// TIA Portal V17 export
// export: Created 2024-08-07T21:44:00.5183403Z, ExportSetting WithDefaults, DisplayName Totally Integrated Automation Portal, DisplayVersion V17 Update 7, DisplayName TIA Portal Openness, DisplayVersion V17 Update 7, DisplayName TIA Portal Version Control Interface, DisplayVersion V17, DisplayName SINAMICS Startdrive Advanced, DisplayVersion V17 SP2, DisplayName SINAMICS Startdrive G110M, G120, G120C, G120D, G120P, G115D, DisplayVersion V17 SP2, DisplayName SINAMICS Startdrive G130, G150, S120, S150, SINAMICS MV, S210, DisplayVersion V17 SP2, DisplayName STEP 7 Professional, DisplayVersion V17 Update 7, DisplayName STEP 7 Safety, DisplayVersion V17 Update 6, DisplayName WinCC Advanced / Unified PC, DisplayVersion V17 Update 7
FUNCTION_BLOCK "FB_DateTimeAndShifts"   // FB5010, LAD
{ S7_Optimized_Access := 'TRUE' }
VERSION : 0.1
// stored: AutoNumber false, IsIECCheckEnabled false, IsRetainMemResEnabled false, MemoryReserve 100, SetENOAutomatically false, UDAEnableTagReadback false
   VAR_INPUT
      iSettingsSecurity : Bool;
   END_VAR
   VAR
      Edges : Struct
         Shift1Started : Bool;
         Shift2Started : Bool;
         Shift3Started : Bool;
      END_STRUCT;
   END_VAR
   VAR RETAIN
      Settings : Struct
         Actual { S7_SetPoint := 'True'} : "UDT_DateTimeAndShiftsSettings";
         Last { S7_SetPoint := 'True'} : "UDT_DateTimeAndShiftsSettings";
         Status : Struct
            SettingsCanBeChanged : Bool;   // 0= No
         END_STRUCT;
         Commands : Struct
            DateAndTimeUse : Bool;
            DateAndTimeSet : Bool;
         END_STRUCT;
      END_STRUCT;
   END_VAR
   VAR
      ActualValues : Struct
         DateAndTime : DTL;
         DayOfYear : UInt;
      END_STRUCT;
      ShiftStatus { S7_SetPoint := 'True'} : "UDT_ShiftStatus";
      TimeTransformationRule { S7_SetPoint := 'True'} : TimeTransformationRule;
      Set_timezone_results { ExternalAccessible := 'False'; ExternalVisible := 'False'; ExternalWritable := 'False'} : Struct
         done { ExternalAccessible := 'False'; ExternalVisible := 'False'; ExternalWritable := 'False'} : Bool;
         busy { ExternalAccessible := 'False'; ExternalVisible := 'False'; ExternalWritable := 'False'} : Bool;
         error { ExternalAccessible := 'False'; ExternalVisible := 'False'; ExternalWritable := 'False'} : Bool;
         status { ExternalAccessible := 'False'; ExternalVisible := 'False'; ExternalWritable := 'False'} : Word;
      END_STRUCT;
   END_VAR
   VAR_TEMP
      i : Int;
      ui : UInt;
      actual_time : Time_Of_Day;
      dst : Bool;
   END_VAR
   VAR_TEMP   // added for the SCL form of the ladder/FBD networks
      _w1 : Bool;
      _w2 : Bool;
      _w3 : Bool;
      _w4 : Bool;
      _w5 : Bool;
      _w6 : Bool;
      _w7 : Bool;
      _w8 : Bool;
   END_VAR
BEGIN

REGION Network 1 (SCL)
   #TimeTransformationRule.Bias := -360;
   #TimeTransformationRule.DaylightBias := 0;
   #TimeTransformationRule.DaylightStartMonth := 3;
   #TimeTransformationRule.DaylightStartWeek := 5;
   #TimeTransformationRule.DaylightStartWeekday := 1;
   #TimeTransformationRule.DaylightStartHour := 2;
   #TimeTransformationRule.DaylightStartMinute := 0;
   #TimeTransformationRule.StandardStartMonth := 10;
   #TimeTransformationRule.StandardStartWeek := 5;
   #TimeTransformationRule.StandardStartWeekday := 1;
   #TimeTransformationRule.StandardStartHour := 3;
   #TimeTransformationRule.StandardStartMinute := 0;
END_REGION

REGION Network 2: Settings control
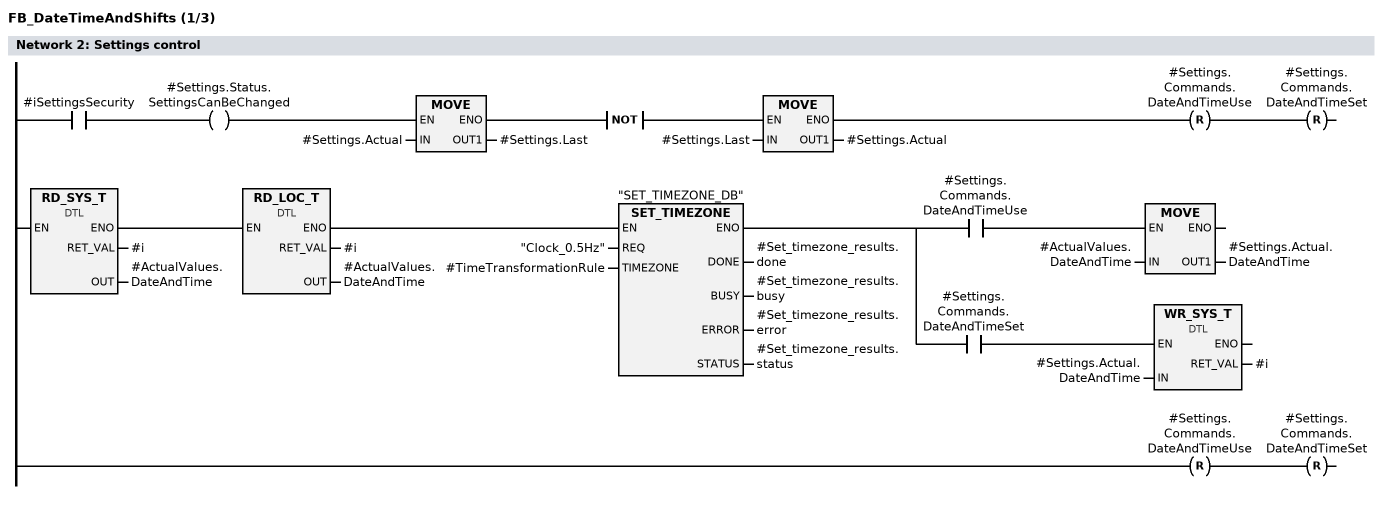
   RUNG wire#powerrail
      Contact( #iSettingsSecurity )
      Coil( #Settings.Status.SettingsCanBeChanged )
      Move(in := #Settings.Actual, out1 => #Settings.Last)
      Not()
      Move(in := #Settings.Last, out1 => #Settings.Actual)
      R_Coil( #Settings.Commands.DateAndTimeUse )
      R_Coil( #Settings.Commands.DateAndTimeSet )
   END_RUNG
   RUNG wire#powerrail
      { S7_Templates := "date_type := DTL" } RD_SYS_T(RET_VAL => #i, OUT => #ActualValues.DateAndTime)
      { S7_Templates := "date_type := DTL" } RD_LOC_T(RET_VAL => #i, OUT => #ActualValues.DateAndTime)
      "SET_TIMEZONE_DB".SET_TIMEZONE(REQ := "Clock_0.5Hz", TimeZone := #TimeTransformationRule, DONE => #Set_timezone_results.done, BUSY => #Set_timezone_results.busy, ERROR => #Set_timezone_results.error, STATUS => #Set_timezone_results.status)
      wire#w1
      Contact( #Settings.Commands.DateAndTimeUse )
      Move(in := #ActualValues.DateAndTime, out1 => #Settings.Actual.DateAndTime)
   END_RUNG
   RUNG wire#w1
      Contact( #Settings.Commands.DateAndTimeSet )
      { S7_Templates := "date_type := DTL" } WR_SYS_T(IN := #Settings.Actual.DateAndTime, RET_VAL => #i)
   END_RUNG
   RUNG wire#powerrail
      R_Coil( #Settings.Commands.DateAndTimeUse )
      R_Coil( #Settings.Commands.DateAndTimeSet )
   END_RUNG
   // the same network as SCL:
   #Settings.Status.SettingsCanBeChanged := #iSettingsSecurity;
   IF #iSettingsSecurity THEN #Settings.Last := #Settings.Actual; END_IF;
   IF NOT #iSettingsSecurity THEN
       #Settings.Actual := #Settings.Last;
       #Settings.Commands.DateAndTimeUse := FALSE;
       #Settings.Commands.DateAndTimeSet := FALSE;
   END_IF;
   #i := RD_SYS_T(OUT => #ActualValues.DateAndTime, ENO => #_w1);
   #i := RD_LOC_T(EN := #_w1, OUT => #ActualValues.DateAndTime, ENO => #_w2);
   "SET_TIMEZONE_DB"(EN := #_w2,   // SET_TIMEZONE
                     REQ := "Clock_0.5Hz",
                     TimeZone := #TimeTransformationRule,
                     DONE => #Set_timezone_results.done,
                     BUSY => #Set_timezone_results.busy,
                     ERROR => #Set_timezone_results.error,
                     STATUS => #Set_timezone_results.status,
                     ENO => #_w3);
   IF #_w3 AND #Settings.Commands.DateAndTimeUse THEN
       #Settings.Actual.DateAndTime := #ActualValues.DateAndTime;
   END_IF;
   IF #_w3 AND #Settings.Commands.DateAndTimeSet THEN
       #i := WR_SYS_T(IN := #Settings.Actual.DateAndTime);
   END_IF;
   #Settings.Commands.DateAndTimeUse := FALSE;
   #Settings.Commands.DateAndTimeSet := FALSE;
END_REGION

REGION Network 3: Day of year
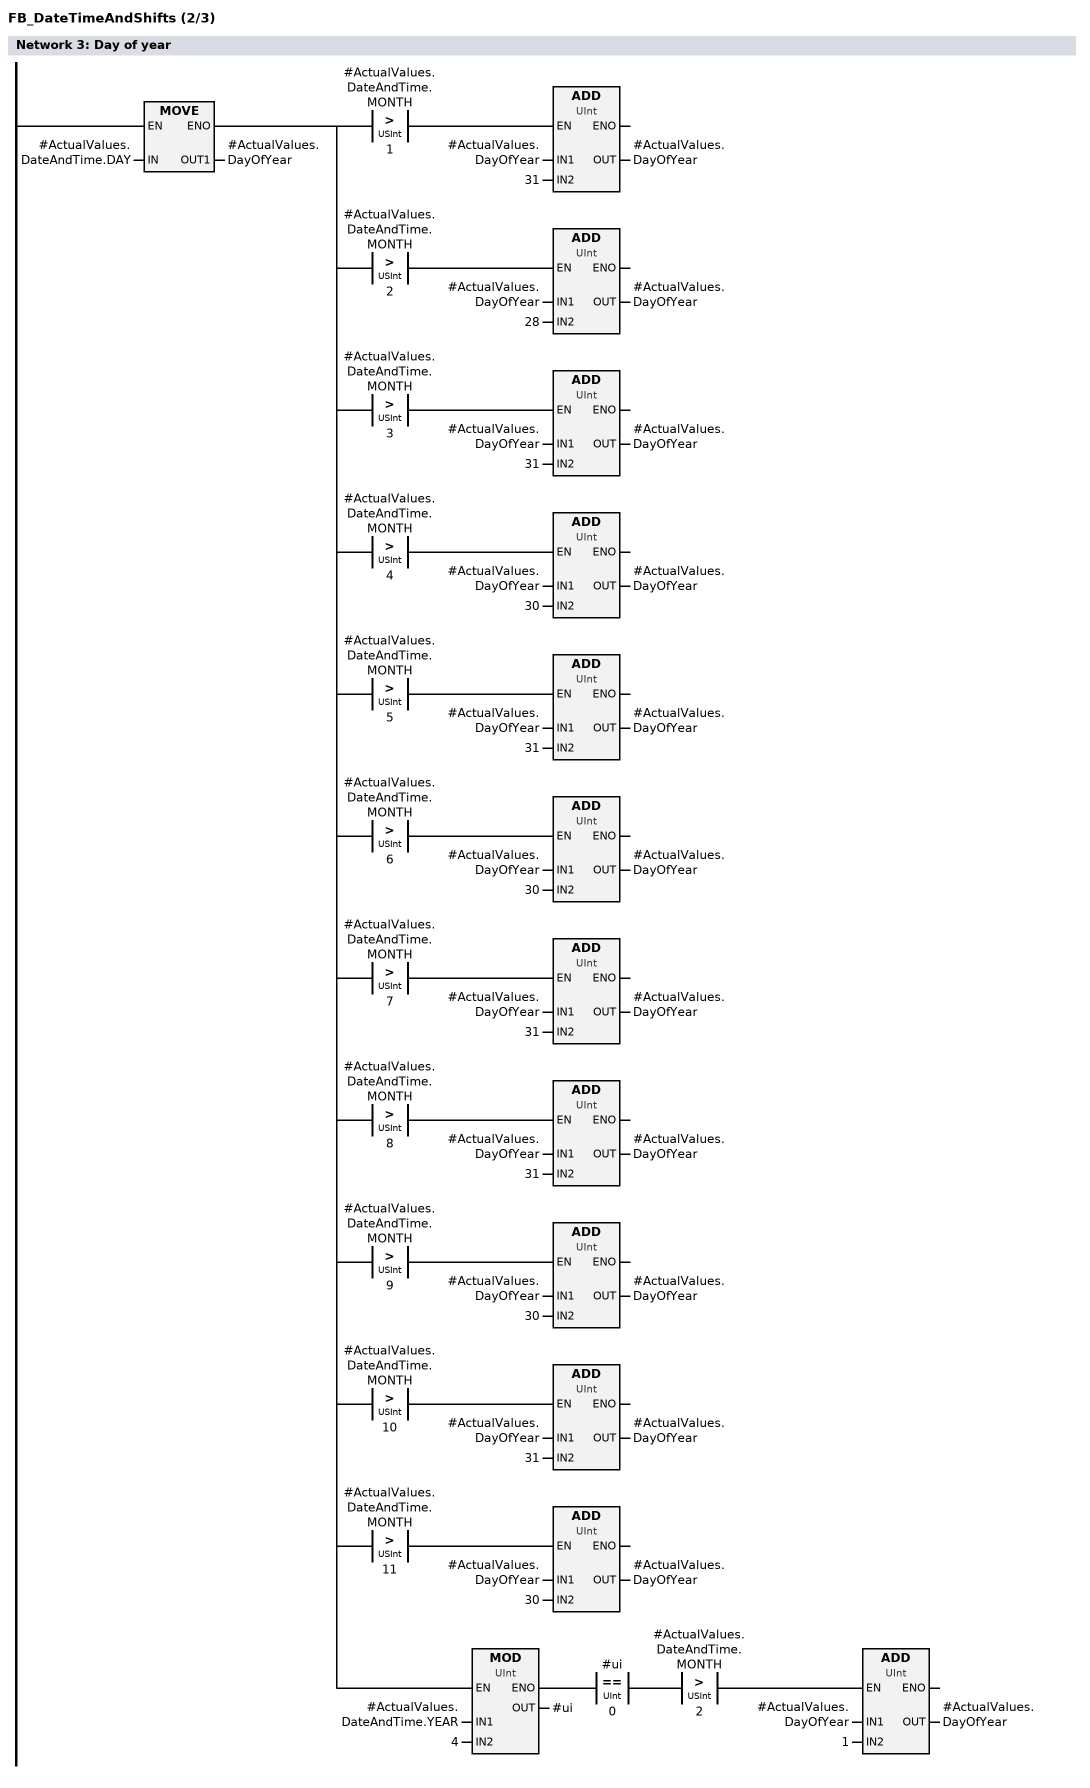
   RUNG wire#powerrail
      Move(in := #ActualValues.DateAndTime.DAY, out1 => #ActualValues.DayOfYear)
      wire#w1
      { S7_Templates := "SrcType := USInt" } GT_Contact(in1 := #ActualValues.DateAndTime.MONTH, in2 := 1)
      { S7_Templates := "SrcType := UInt" } Add(in1 := #ActualValues.DayOfYear, in2 := 31, out => #ActualValues.DayOfYear)
   END_RUNG
   RUNG wire#w1
      { S7_Templates := "SrcType := USInt" } GT_Contact(in1 := #ActualValues.DateAndTime.MONTH, in2 := 2)
      { S7_Templates := "SrcType := UInt" } Add(in1 := #ActualValues.DayOfYear, in2 := 28, out => #ActualValues.DayOfYear)
   END_RUNG
   RUNG wire#w1
      { S7_Templates := "SrcType := USInt" } GT_Contact(in1 := #ActualValues.DateAndTime.MONTH, in2 := 3)
      { S7_Templates := "SrcType := UInt" } Add(in1 := #ActualValues.DayOfYear, in2 := 31, out => #ActualValues.DayOfYear)
   END_RUNG
   RUNG wire#w1
      { S7_Templates := "SrcType := USInt" } GT_Contact(in1 := #ActualValues.DateAndTime.MONTH, in2 := 4)
      { S7_Templates := "SrcType := UInt" } Add(in1 := #ActualValues.DayOfYear, in2 := 30, out => #ActualValues.DayOfYear)
   END_RUNG
   RUNG wire#w1
      { S7_Templates := "SrcType := USInt" } GT_Contact(in1 := #ActualValues.DateAndTime.MONTH, in2 := 5)
      { S7_Templates := "SrcType := UInt" } Add(in1 := #ActualValues.DayOfYear, in2 := 31, out => #ActualValues.DayOfYear)
   END_RUNG
   RUNG wire#w1
      { S7_Templates := "SrcType := USInt" } GT_Contact(in1 := #ActualValues.DateAndTime.MONTH, in2 := 6)
      { S7_Templates := "SrcType := UInt" } Add(in1 := #ActualValues.DayOfYear, in2 := 30, out => #ActualValues.DayOfYear)
   END_RUNG
   RUNG wire#w1
      { S7_Templates := "SrcType := USInt" } GT_Contact(in1 := #ActualValues.DateAndTime.MONTH, in2 := 7)
      { S7_Templates := "SrcType := UInt" } Add(in1 := #ActualValues.DayOfYear, in2 := 31, out => #ActualValues.DayOfYear)
   END_RUNG
   RUNG wire#w1
      { S7_Templates := "SrcType := USInt" } GT_Contact(in1 := #ActualValues.DateAndTime.MONTH, in2 := 8)
      { S7_Templates := "SrcType := UInt" } Add(in1 := #ActualValues.DayOfYear, in2 := 31, out => #ActualValues.DayOfYear)
   END_RUNG
   RUNG wire#w1
      { S7_Templates := "SrcType := USInt" } GT_Contact(in1 := #ActualValues.DateAndTime.MONTH, in2 := 9)
      { S7_Templates := "SrcType := UInt" } Add(in1 := #ActualValues.DayOfYear, in2 := 30, out => #ActualValues.DayOfYear)
   END_RUNG
   RUNG wire#w1
      { S7_Templates := "SrcType := USInt" } GT_Contact(in1 := #ActualValues.DateAndTime.MONTH, in2 := 10)
      { S7_Templates := "SrcType := UInt" } Add(in1 := #ActualValues.DayOfYear, in2 := 31, out => #ActualValues.DayOfYear)
   END_RUNG
   RUNG wire#w1
      { S7_Templates := "SrcType := USInt" } GT_Contact(in1 := #ActualValues.DateAndTime.MONTH, in2 := 11)
      { S7_Templates := "SrcType := UInt" } Add(in1 := #ActualValues.DayOfYear, in2 := 30, out => #ActualValues.DayOfYear)
   END_RUNG
   RUNG wire#w1
      { S7_Templates := "SrcType := UInt" } Mod(in1 := #ActualValues.DateAndTime.YEAR, in2 := 4, out => #ui)
      { S7_Templates := "SrcType := UInt" } EQ_Contact(in1 := #ui, in2 := 0)
      { S7_Templates := "SrcType := USInt" } GT_Contact(in1 := #ActualValues.DateAndTime.MONTH, in2 := 2)
      { S7_Templates := "SrcType := UInt" } Add(in1 := #ActualValues.DayOfYear, in2 := 1, out => #ActualValues.DayOfYear)
   END_RUNG
   // the same network as SCL:
   #ActualValues.DayOfYear := #ActualValues.DateAndTime.DAY;
   IF #ActualValues.DateAndTime.MONTH > 1 THEN
       #ActualValues.DayOfYear := #ActualValues.DayOfYear + 31;
   END_IF;
   IF #ActualValues.DateAndTime.MONTH > 2 THEN
       #ActualValues.DayOfYear := #ActualValues.DayOfYear + 28;
   END_IF;
   IF #ActualValues.DateAndTime.MONTH > 3 THEN
       #ActualValues.DayOfYear := #ActualValues.DayOfYear + 31;
   END_IF;
   IF #ActualValues.DateAndTime.MONTH > 4 THEN
       #ActualValues.DayOfYear := #ActualValues.DayOfYear + 30;
   END_IF;
   IF #ActualValues.DateAndTime.MONTH > 5 THEN
       #ActualValues.DayOfYear := #ActualValues.DayOfYear + 31;
   END_IF;
   IF #ActualValues.DateAndTime.MONTH > 6 THEN
       #ActualValues.DayOfYear := #ActualValues.DayOfYear + 30;
   END_IF;
   IF #ActualValues.DateAndTime.MONTH > 7 THEN
       #ActualValues.DayOfYear := #ActualValues.DayOfYear + 31;
   END_IF;
   IF #ActualValues.DateAndTime.MONTH > 8 THEN
       #ActualValues.DayOfYear := #ActualValues.DayOfYear + 31;
   END_IF;
   IF #ActualValues.DateAndTime.MONTH > 9 THEN
       #ActualValues.DayOfYear := #ActualValues.DayOfYear + 30;
   END_IF;
   IF #ActualValues.DateAndTime.MONTH > 10 THEN
       #ActualValues.DayOfYear := #ActualValues.DayOfYear + 31;
   END_IF;
   IF #ActualValues.DateAndTime.MONTH > 11 THEN
       #ActualValues.DayOfYear := #ActualValues.DayOfYear + 30;
   END_IF;
   #ui := #ActualValues.DateAndTime.YEAR MOD 4;
   IF (#ui = 0) AND (#ActualValues.DateAndTime.MONTH > 2) THEN
       #ActualValues.DayOfYear := #ActualValues.DayOfYear + 1;
   END_IF;
END_REGION

REGION Network 4: Shifts
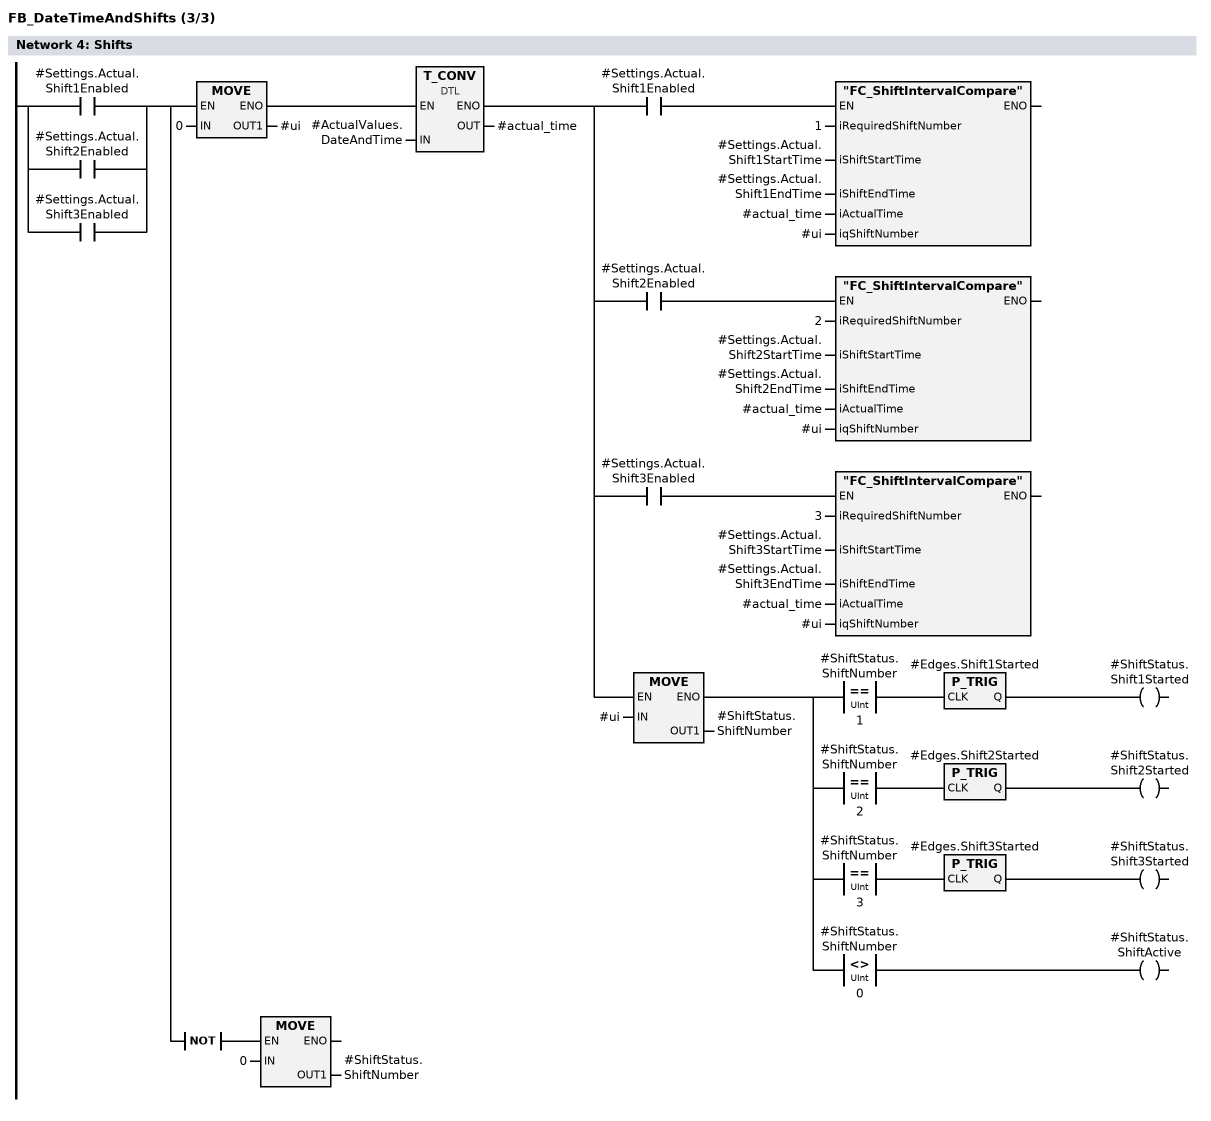
   RUNG wire#powerrail
      Contact( #Settings.Actual.Shift1Enabled )
      wire#w1
      Move(in := 0, out1 => #ui)
      { S7_Templates := "[src_type := DTL, dest_type := Time_Of_Day]" } T_CONV(IN := #ActualValues.DateAndTime, OUT => #actual_time)
      wire#w2
      Contact( #Settings.Actual.Shift1Enabled )
      "FC_ShiftIntervalCompare"(iRequiredShiftNumber := 1, iShiftStartTime := #Settings.Actual.Shift1StartTime, iShiftEndTime := #Settings.Actual.Shift1EndTime, iActualTime := #actual_time, iqShiftNumber := #ui)
   END_RUNG
   RUNG wire#powerrail
      Contact( #Settings.Actual.Shift2Enabled )
   END_RUNG wire#w1
   RUNG wire#powerrail
      Contact( #Settings.Actual.Shift3Enabled )
   END_RUNG wire#w1
   RUNG wire#w2
      Contact( #Settings.Actual.Shift2Enabled )
      "FC_ShiftIntervalCompare"(iRequiredShiftNumber := 2, iShiftStartTime := #Settings.Actual.Shift2StartTime, iShiftEndTime := #Settings.Actual.Shift2EndTime, iActualTime := #actual_time, iqShiftNumber := #ui)
   END_RUNG
   RUNG wire#w2
      Contact( #Settings.Actual.Shift3Enabled )
      "FC_ShiftIntervalCompare"(iRequiredShiftNumber := 3, iShiftStartTime := #Settings.Actual.Shift3StartTime, iShiftEndTime := #Settings.Actual.Shift3EndTime, iActualTime := #actual_time, iqShiftNumber := #ui)
   END_RUNG
   RUNG wire#w2
      Move(in := #ui, out1 => #ShiftStatus.ShiftNumber)
      wire#w3
      { S7_Templates := "SrcType := UInt" } EQ_Contact(in1 := #ShiftStatus.ShiftNumber, in2 := 1)
      P_Trig( #Edges.Shift1Started )
      Coil( #ShiftStatus.Shift1Started )
   END_RUNG
   RUNG wire#w3
      { S7_Templates := "SrcType := UInt" } EQ_Contact(in1 := #ShiftStatus.ShiftNumber, in2 := 2)
      P_Trig( #Edges.Shift2Started )
      Coil( #ShiftStatus.Shift2Started )
   END_RUNG
   RUNG wire#w3
      { S7_Templates := "SrcType := UInt" } EQ_Contact(in1 := #ShiftStatus.ShiftNumber, in2 := 3)
      P_Trig( #Edges.Shift3Started )
      Coil( #ShiftStatus.Shift3Started )
   END_RUNG
   RUNG wire#w3
      { S7_Templates := "SrcType := UInt" } NE_Contact(in1 := #ShiftStatus.ShiftNumber, in2 := 0)
      Coil( #ShiftStatus.ShiftActive )
   END_RUNG
   RUNG wire#w1
      Not()
      Move(in := 0, out1 => #ShiftStatus.ShiftNumber)
   END_RUNG
   // the same network as SCL:
   #_w1 := #Settings.Actual.Shift1Enabled OR #Settings.Actual.Shift2Enabled OR #Settings.Actual.Shift3Enabled;
   IF #_w1 THEN #ui := 0; END_IF;
   T_CONV(EN := #_w1, IN := #ActualValues.DateAndTime, OUT => #actual_time, ENO => #_w2);
   IF #_w2 AND #Settings.Actual.Shift1Enabled THEN
       "FC_ShiftIntervalCompare"(iRequiredShiftNumber := 1,
                               iShiftStartTime := #Settings.Actual.Shift1StartTime,
                               iShiftEndTime := #Settings.Actual.Shift1EndTime,
                               iActualTime := #actual_time,
                               iqShiftNumber := #ui);
   END_IF;
   IF #_w2 AND #Settings.Actual.Shift2Enabled THEN
       "FC_ShiftIntervalCompare"(iRequiredShiftNumber := 2,
                               iShiftStartTime := #Settings.Actual.Shift2StartTime,
                               iShiftEndTime := #Settings.Actual.Shift2EndTime,
                               iActualTime := #actual_time,
                               iqShiftNumber := #ui);
   END_IF;
   IF #_w2 AND #Settings.Actual.Shift3Enabled THEN
       "FC_ShiftIntervalCompare"(iRequiredShiftNumber := 3,
                               iShiftStartTime := #Settings.Actual.Shift3StartTime,
                               iShiftEndTime := #Settings.Actual.Shift3EndTime,
                               iActualTime := #actual_time,
                               iqShiftNumber := #ui);
   END_IF;
   IF #_w2 THEN #ShiftStatus.ShiftNumber := #ui; END_IF;
   #_w3 := #_w2 AND (#ShiftStatus.ShiftNumber = 1);
   #_w4 := #_w3 AND NOT #Edges.Shift1Started;   // rising edge
   #Edges.Shift1Started := #_w3;
   #ShiftStatus.Shift1Started := #_w4;
   #_w5 := #_w2 AND (#ShiftStatus.ShiftNumber = 2);
   #_w6 := #_w5 AND NOT #Edges.Shift2Started;   // rising edge
   #Edges.Shift2Started := #_w5;
   #ShiftStatus.Shift2Started := #_w6;
   #_w7 := #_w2 AND (#ShiftStatus.ShiftNumber = 3);
   #_w8 := #_w7 AND NOT #Edges.Shift3Started;   // rising edge
   #Edges.Shift3Started := #_w7;
   #ShiftStatus.Shift3Started := #_w8;
   #ShiftStatus.ShiftActive := #_w2 AND (#ShiftStatus.ShiftNumber <> 0);
   IF NOT #_w1 THEN #ShiftStatus.ShiftNumber := 0; END_IF;
END_REGION
END_FUNCTION_BLOCK
